TYPE ST_SYMBOL_AddressInfo :	(* 8 bytes *)
STRUCT
	pSymAddr	: 	DWORD;
	nSymSize	:	UDINT;
END_STRUCT
END_TYPE

(* stored: Version 1.1.0.1, ProductVersion 3.1.4024.15
   DUT ST_SYMBOL_AddressInfo: Id {9006efdc-eda8-433c-8f4b-e820ae66c5e6} *)
